// TIA Portal V20 export
// export: Created 2026-04-28T10:17:59.5077277Z, ExportSetting WithDefaults, DisplayName Totally Integrated Automation Portal, DisplayVersion V20, DisplayName TIA Portal Openness, DisplayVersion V20, DisplayName TIA Portal Version Control Interface, DisplayVersion V20, DisplayName SINAMICS Startdrive Advanced, DisplayVersion V20, DisplayName SINAMICS Startdrive G130, G150, S120, S150, SINAMICS MV, G220, S200, S210, DisplayVersion V20, DisplayName SINAMICS Startdrive G110M, G120, G120C, G120D, G120P, G115D, DisplayVersion V20, DisplayName STEP 7 Professional, DisplayVersion V20, DisplayName STEP 7 Safety, DisplayVersion V20, DisplayName WinCC Basic/Comfort/Advanced, DisplayVersion V20, DisplayName WinCC Unified, DisplayVersion V20
VAR_GLOBAL   // PLC tag table "Standard-Variablentabelle"
   xtest1 AT %M499.0 : Bool;   // Test1
   System_Byte AT %MB1 : Byte;
   Clock_Byte AT %MB5 : Byte;
   diEnable AT %I25.0 : Bool;   // Sperren
   Tag_1 AT %M854.1 : Bool;
   Tag_2 AT %M854.2 : Bool;
   aiSlPre AT %MW36 : Word;
   TO_Drive_Main_Fan_Actor_Interface_AddressIn AT %I256.0 : "PD_TEL1_IN";
   TO_Drive_Powder_Return_Fan_Actor_Interface_AddressIn AT %I260.0 : "PD_TEL1_IN";
   TO_Drive_Slip_Pump_Actor_Interface_AddressIn AT %I264.0 : "PD_TEL1_IN";
   diVaSwFlapOpen AT %I24.7 : Bool;   // Ventil Umschaltung Klappe öffnen
   diVaSwFlapClose AT %I24.6 : Bool;   // Ventil Umschaltung Klappe schliessen
   TO_Drive_Main_Fan_Actor_Interface_AddressOut AT %Q256.0 : "PD_TEL1_OUT";
   TO_Drive_Powder_Return_Fan_Actor_Interface_AddressOut AT %Q260.0 : "PD_TEL1_OUT";
   TO_Drive_Slip_Pump_Actor_Interface_AddressOut AT %Q264.0 : "PD_TEL1_OUT";
   Tag_3 AT %I67.0 : Bool;
   Tag_4 AT %I67.1 : Bool;
   Tag_5 AT %I67.2 : Bool;
   Tag_6 AT %I67.3 : Bool;
   Tag_7 AT %I74.0 : Bool;
   Tag_8 AT %I74.1 : Bool;
   Tag_9 AT %I74.2 : Bool;
   Tag_10 AT %I74.3 : Bool;
   Tag_11 AT %I74.4 : Bool;
   Tag_12 AT %I74.6 : Bool;
END_VAR
